PROGRAM AS101
VAR
	PUMPMOTION: fbPumpMotion;
	WATCHDOG: fbWatchdogSwitching;
	RST: fbResetButton;
	CBL: fbFirealarm;
	AUT: fbFusealarm;
	JFB: fbJfb;
	OSP: fbOvervoltageProtection;
	MODBUS: fbModbusSekvensArray;
	SYSTEM: fbOaksSystem;
	TCH1: fbTimeChannelWp;
	TCH2: fbTimeChannelWp;
	ODT: fbReadAdsRealOutdoorMeantempWp_STL;	
	FASBROTT: fbDigitalAlarmIO;		
	ASTRO: fbSunClock := (SP1 := 57.7089, SP2 := 11.9746); 
	F_trigVentilmotion: F_TRIG;
	TOF_Ventilmotion: TOF;		

END_VAR
VAR_OUTPUT
	TCH1_bOutput AT %Q* : BOOL; //Tidkanal 1
	TCH2_bOutput AT %Q* : BOOL; //Tidkanal 2
	bVentilmotion: BOOL; //Ventilmotion aktiv~wp:[trendoptions]i:14400, t:1	
	FASBROTT_AL:BOOL; //larm fasbrottsrelä~wp:
	

END_VAR
VAR PERSISTENT

END_VAR

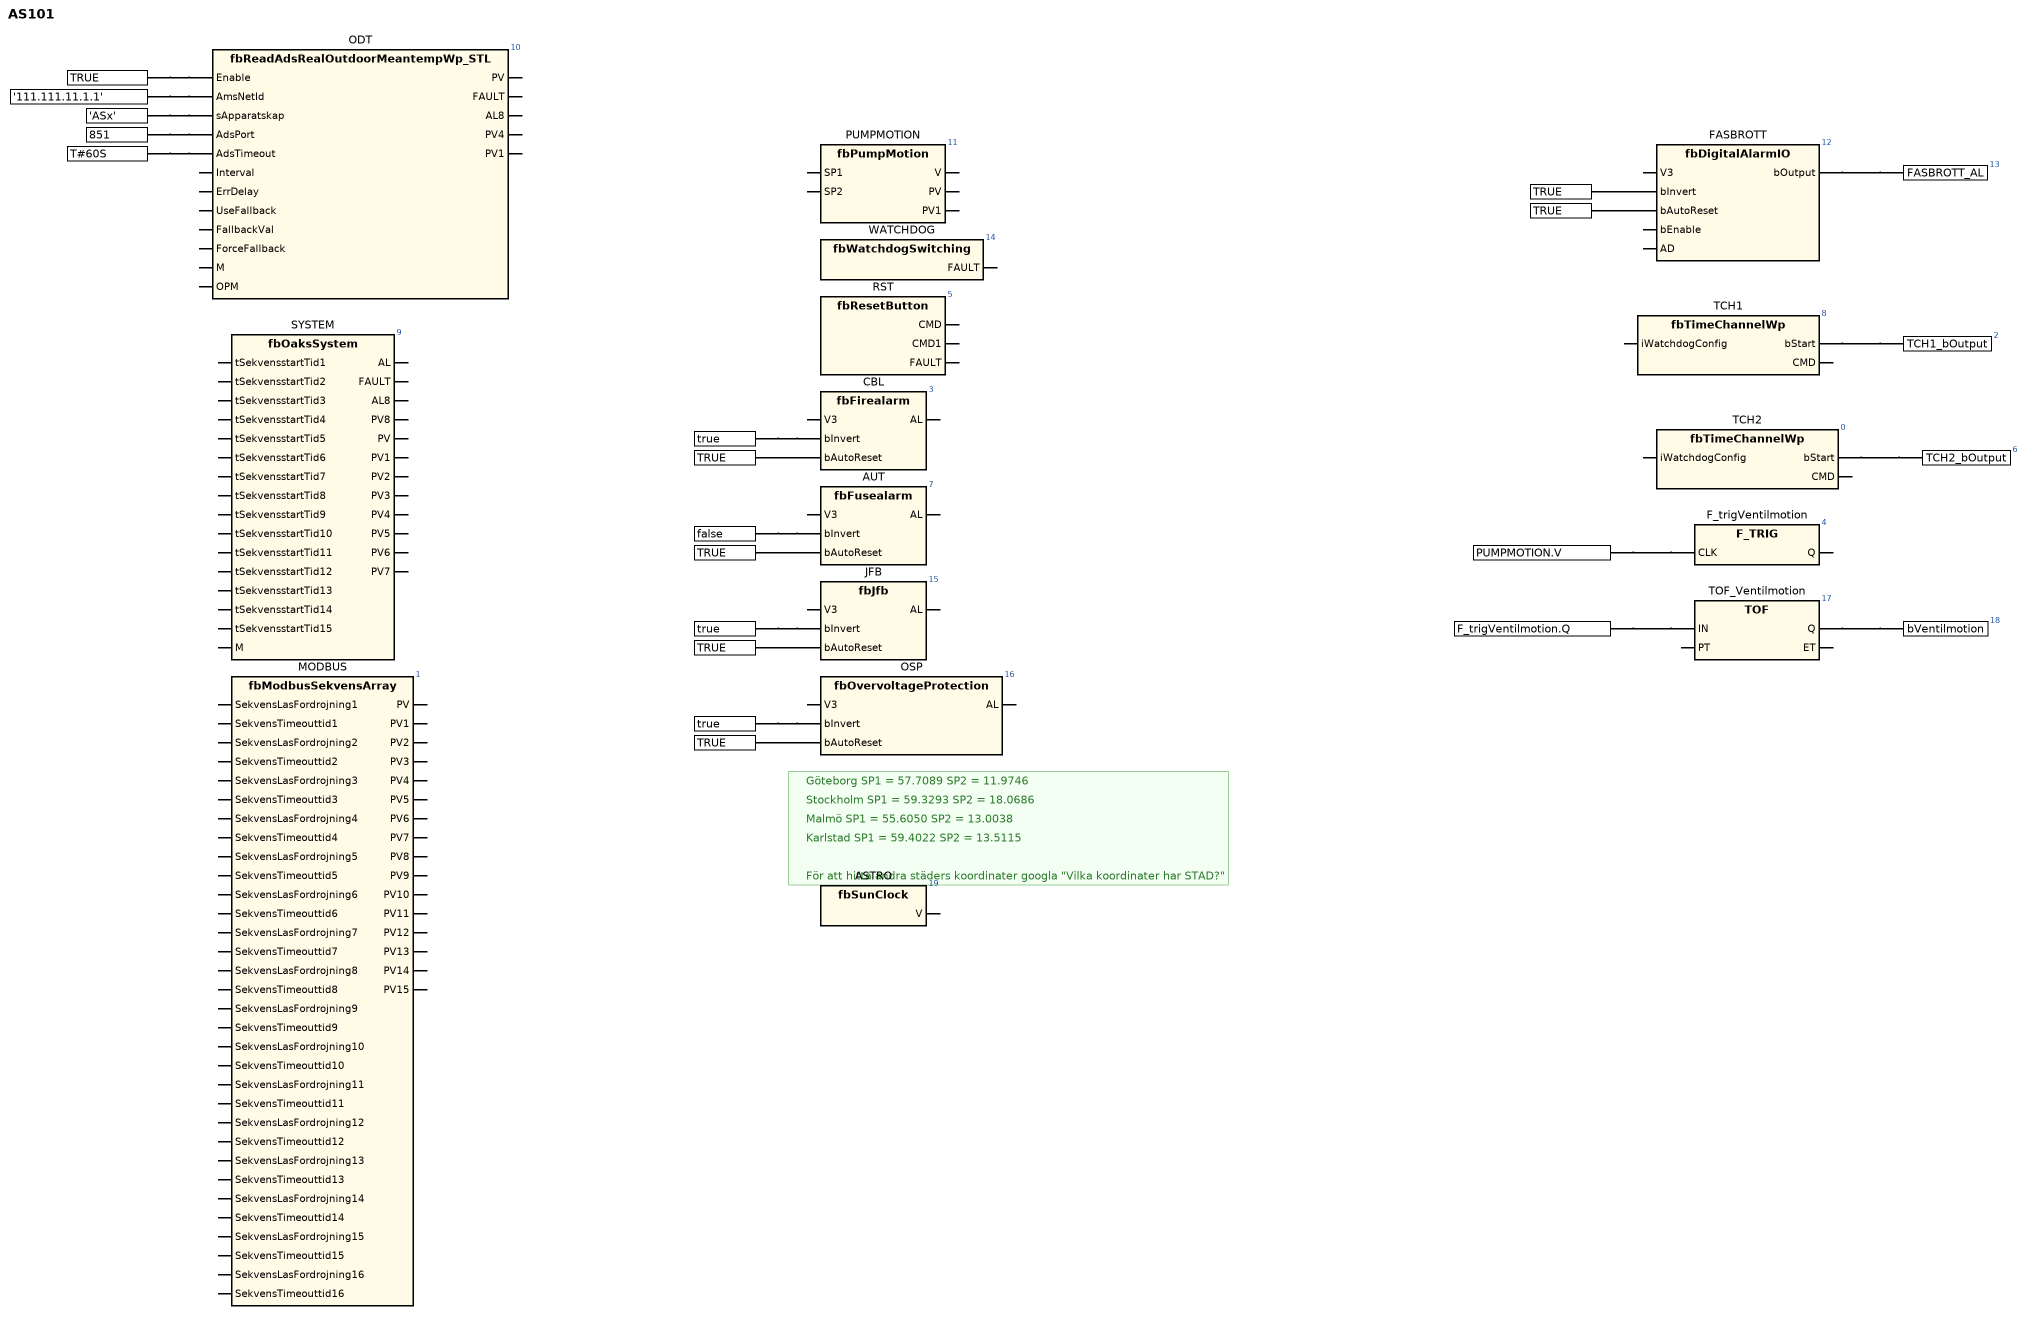
TCH2(); // fbTimeChannelWp
MODBUS(); // fbModbusSekvensArray
TCH1_bOutput := TCH1.bStart;
CBL(bInvert := true, bAutoReset := TRUE); // fbFirealarm
F_trigVentilmotion(CLK := PUMPMOTION.V); // F_TRIG
RST(); // fbResetButton
TCH2_bOutput := TCH2.bStart;
AUT(bInvert := false, bAutoReset := TRUE); // fbFusealarm
TCH1(); // fbTimeChannelWp
SYSTEM(); // fbOaksSystem
ODT(Enable := TRUE, AmsNetId := '111.111.11.1.1', sApparatskap := 'ASx', AdsPort := 851, AdsTimeout := T#60S); // fbReadAdsRealOutdoorMeantempWp_STL
PUMPMOTION(); // fbPumpMotion
FASBROTT(bInvert := TRUE, bAutoReset := TRUE); // fbDigitalAlarmIO
FASBROTT_AL := FASBROTT.bOutput;
WATCHDOG(); // fbWatchdogSwitching
JFB(bInvert := true, bAutoReset := TRUE); // fbJfb
OSP(bInvert := true, bAutoReset := TRUE); // fbOvervoltageProtection
TOF_Ventilmotion(IN := F_trigVentilmotion.Q); // TOF
bVentilmotion := TOF_Ventilmotion.Q;
// 		Göteborg SP1 = 57.7089 SP2 = 11.9746
// 		Stockholm SP1 = 59.3293 SP2 = 18.0686
// 		Malmö SP1 = 55.6050 SP2 = 13.0038
// 		Karlstad SP1 = 59.4022 SP2 = 13.5115
//
// 		För att hitta andra städers koordinater googla "Vilka koordinater har STAD?"
ASTRO(); // fbSunClock

END_PROGRAM

(* stored: Version 1.1.0.1, ProductVersion 3.1.4024.13
   POU AS101: Id {27438f4d-ba85-41de-bb61-3ac6d62d36f6}, SpecialFunc None *)
